{attribute 'no-analysis'}
TYPE ST_EL3446_VariantValues :
STRUCT
	astIx 			: ARRAY[1..6] OF ST_EL3446_VariantIx;
END_STRUCT
END_TYPE

(* stored: Version 1.1.0.1, ProductVersion 3.1.4024.12
   DUT ST_EL3446_VariantValues: Id {fb56ac51-7081-4ec2-9818-7a4a65f07349} *)
